
FUNCTION CB_le_date : BOOL


TITLE = ' Test Whether IN0 is lower than or equal to IN1 '
VERSION : '1.0'
AUTHOR  : CB
NAME    : le_date
FAMILY  : TNI

VAR_INPUT
    IN0 : DATE;
    IN1 : DATE;
END_VAR

BEGIN

CB_le_date := (IN0 <= IN1);

END_FUNCTION
